TYPE TcoAoConfig :
STRUCT
	RawLow:DINT;
	RawHigh:DINT;
	RealLow:REAL;
	RealHigh:REAL;
	Gain: REAL := 1.0;
	Offset: REAL := 0.0;  	

END_STRUCT
END_TYPE

(* stored: Version 1.1.0.1, ProductVersion 3.1.4024.9
   DUT TcoAoConfig: Id {1ebf84b8-fca2-08b7-1e0c-0be1a3bc934d} *)
